TYPE "Ttest"
TITLE = Ttest_udt
VERSION : 0.1
//Typ danych będący interfacem do ruchów w trybie ręcznym
   STRUCT
      fp_HP : Bool;
      fp_WP : Bool;
      fp_IDLE : Bool;
      WP_on : Bool;
      dummy_HP : Bool;
      dummy_WP : Bool;
      dummy_IDLE : Bool;
      dummy_BRAKE : Bool;
   END_STRUCT;

END_TYPE

